(* PLC project Unnamed, Unknown Unnamed 1 *)
(* stored: creationDateTime 2019-08-06T14:23:42, modificationDateTime 2026-03-16T18:31:36 *)

FUNCTION_BLOCK PumpControl
  VAR_INPUT
    Pump : HMI_NODE := 1;
  END_VAR
  VAR
    strout : HMI_STRING;
  END_VAR
  VAR_INPUT
    strin : HMI_STRING := blup;
  END_VAR

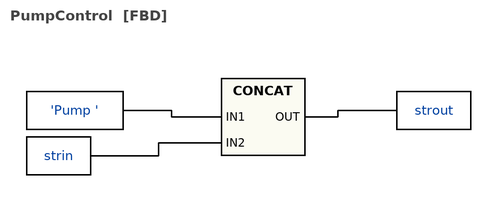
(* FBD diagram, written out as Structured Text *)
strout := CONCAT('Pump ', strin);
END_FUNCTION_BLOCK

PROGRAM MainStuff
  VAR
    Pump0 : PumpControl;
    Pump1 : PumpControl;
    Pump2 : PumpControl;
    Pump3 : PumpControl;
    Pump4 : PumpControl;
    Pump5 : PumpControl;
    Pump6 : PumpControl;
    Pump7 : PumpControl;
  END_VAR

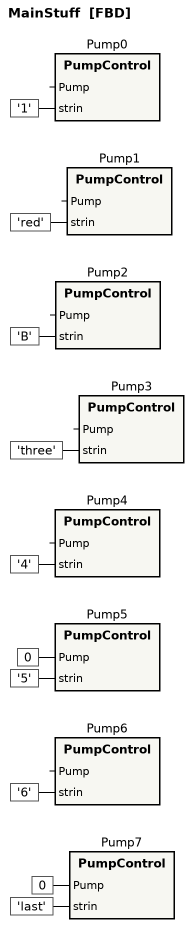
(* FBD diagram, written out as Structured Text *)
Pump0(strin := '1');
Pump1(strin := 'red');
Pump2(strin := 'B');
Pump3(strin := 'three');
Pump4(strin := '4');
Pump5(Pump := 0, strin := '5');
Pump6(strin := '6');
Pump7(Pump := 0, strin := 'last');
END_PROGRAM

CONFIGURATION config
  RESOURCE resource1 ON PLC
    TASK task0(INTERVAL := T#20ms, PRIORITY := 0);
    PROGRAM instance0 WITH task0 : MainStuff;
  END_RESOURCE
END_CONFIGURATION
